Staubli VAL3: stop.pgx

program stop()
  local joint l_jHere
  local string l_sToolStatus
begin
  //
  l_sToolStatus=""
  //
  cls()
  gotoxy(10,6)
  put("Application Ending")
  //
  stopMove()
  resetMotion()
  disablePower()
  // Stop all tasks
  taskKill("TransferQueue1")
  taskKill("overflowPick")
  taskKill("productionCycle")
  taskKill("blow")
  taskKill("changePallet")
  taskKill("isInSafetyArea")
  taskKill("fRobot2sRobot")
  taskKill("robot2PLC")

  if _bConvExist
    call mot:kill()
  endIf

  //
  // Stop conveyor speed
  call setConvSpeed(0,0)
  //
  // Reset triggers
  //  dioSet(dTrigger,0)
  //
  resetMotion()
  //
  //
  // Move up axis 3
  l_jHere=herej()
  l_jHere.j3=90
  //movej(l_jHere,flange,mSlow)
  //
  // Drop the part on the tool
  if bPickDetection
    call getToolStatus(l_sToolStatus)
  endIf
  if l_sToolStatus=="PartInTool" or !bPickDetection
    //movej(jDropPart,flange,mSlow)
    //waitEndMove()
    dBlow=true
    dVacuum=false
    delay(0.5)
    dBlow=false
  else
    dVacuum=false
    dBlow=false
  endIf
  //
  // Go to park position
  //movej(jPark,flange,mSlow)
  //waitEndMove()
  disablePower()
  //
  cls()
  gotoxy(10,6)
  put("Application Ended")
  //
end
